INTERFACE I_InputSourceHistorical EXTENDS I_InputSource

METHOD HistoricalCtrl : BOOL
VAR_INPUT
	stCtrl: REFERENCE TO ST_HMI_InputSourceCtrl;
	stHistStreamInfo: REFERENCE TO ST_HMI_DataSourceHist;
	stRecordInfo: REFERENCE TO ST_HMI_DataSourceHistRecordInfo;
END_VAR
END_METHOD

METHOD UpdateRecordList : BOOL
VAR_INPUT
	sStreamSystemID: GUID;
	stHistStreamInfo: REFERENCE TO ST_HMI_DataSourceHist;
END_VAR
END_METHOD

PROPERTY bCtrlChanged : BOOL
GET
END_GET
END_PROPERTY

END_INTERFACE

(* stored: Itf I_InputSourceHistorical: Id 645ecb90-1f81-443d-b75f-a09d406e0b80
   Method HistoricalCtrl: Id 41ae363a-5533-4b76-84fd-cd047f546f93
   Method UpdateRecordList: Id 7b9143b4-fbc0-46f6-afba-2735bcb16ea2
   Property bCtrlChanged: Id 5cd23029-b103-481f-a181-b81e2d760a70
   Get Get: Id 16f1a860-a4bb-4799-8232-d9398248fc90 *)
